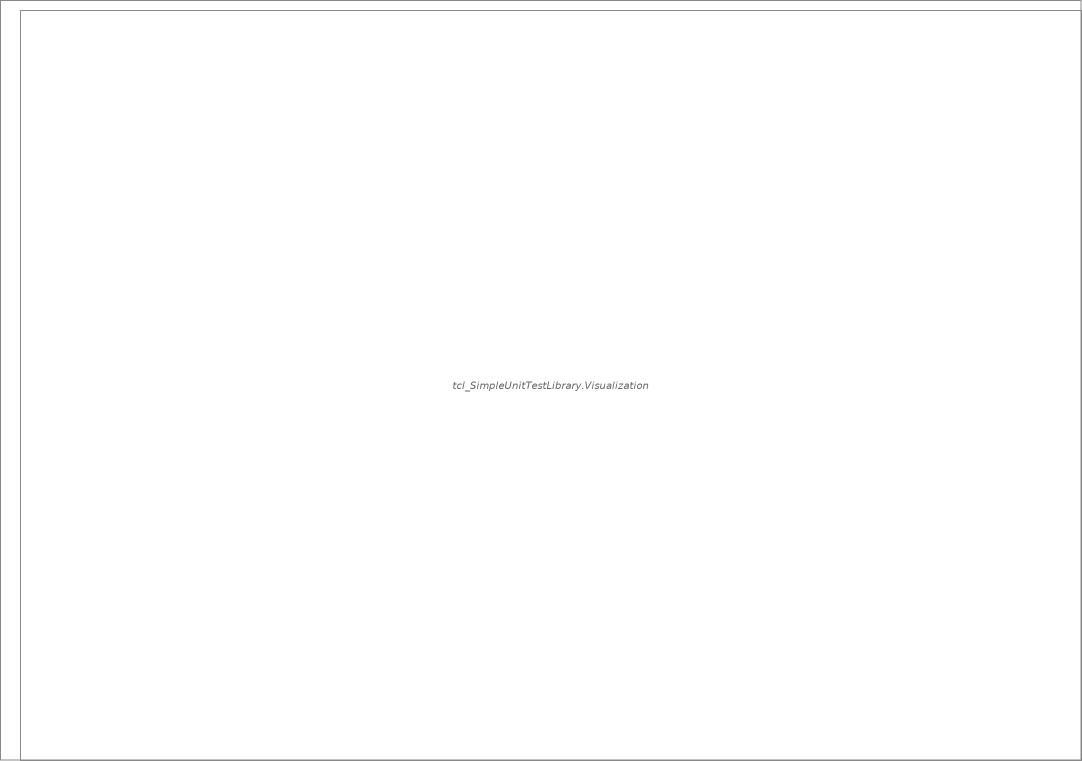
VISUALIZATION Visualization  // 1082x761
    Frame (20,10 1062x751)
        shows tcl_SimpleUnitTestLibrary.Visualization()
END_VISUALIZATION

(* stored: Version 1.1.0.1, ProductVersion 3.1.4024.3
   Visu Visualization: Id {fd9c10a1-8fa5-40cb-94e9-384a02350ea1} *)
